// Mitsubishi GX Works2 project: 21-05-2020 Double outputs   PLC: FX3G

PROGRAM MAIN
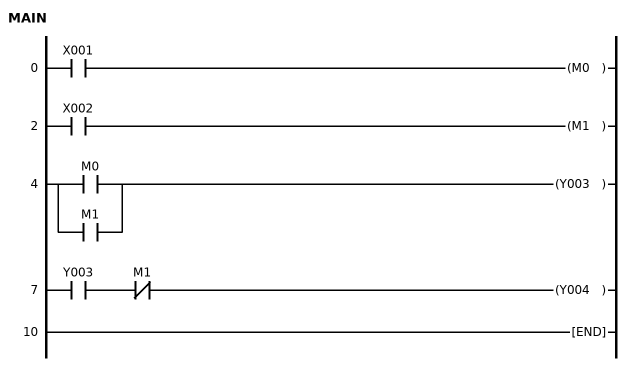
0     LD      X001
      OUT     M0
2     LD      X002
      OUT     M1
4     LD      M0
      OR      M1
      OUT     Y003
7     LD      Y003
      ANI     M1
      OUT     Y004
10    END
END_PROGRAM
